(*
SPDX-FileCopyrightText: © 2026 Oleksandr Tiutyk <trofimich@gmail.com>
SPDX-License-Identifier: MIT
License: https://opensource.org/license/mit
*)

TYPE GENERIC_KEY_VALUE_PAIR :
STRUCT
	Key : GENERIC_VALUE;
	Value : GENERIC_VALUE;
END_STRUCT
END_TYPE

(* stored: Version 1.1.0.1
   DUT GENERIC_KEY_VALUE_PAIR: Id {a21052cd-0952-44b7-848a-1c3c44857d19} *)
